// TIA Portal V17 export
// export: Created 2025-01-08T13:55:36.5022133Z, ExportSetting WithDefaults, DisplayName Totally Integrated Automation Portal, DisplayVersion V17, DisplayName TIA Portal Openness, DisplayVersion V17, DisplayName TIA Portal Version Control Interface, DisplayVersion V17, DisplayName SINAMICS Startdrive Advanced, DisplayVersion V17 Update2, DisplayName SINAMICS Startdrive G130, G150, S120, S150, SINAMICS MV, S210, DisplayVersion V17 Update2, DisplayName SINAMICS Startdrive G110M, G120, G120C, G120D, G120P, G115D, DisplayVersion V17 Update2, DisplayName STEP 7 Professional, DisplayVersion V17, DisplayName STEP 7 Safety, DisplayVersion V17, DisplayName WinCC Advanced, DisplayVersion V17
TYPE "HSMConfigAndMachineParameterMask"
// stored: IsFailsafeCompliant false
   STRUCT
      HSMConfig_1 : "HSMConfigParaMask1";
      HSMConfig_2 : "HSMConfigParaMask2";
      HSMMachine_1 { S7_SetPoint := 'True'} : "HSMMachineParaMask1";
      HSMMachine_2 { S7_SetPoint := 'True'} : "HSMMachineParaMask2";
      HSMMachine_3 { S7_SetPoint := 'True'} : "HSMMachineParaMask3";
      HSMMachine_4 { S7_SetPoint := 'True'} : "HSMMachineParaMask4";
      HSMMachine_5 { S7_SetPoint := 'True'} : "HSMMachineParaMask5";
      HSMMachine_6 { S7_SetPoint := 'True'} : "HSMMachineParaMask6";
      HSMMachine_7 { S7_SetPoint := 'True'} : "HSMMachineParaMask7";
      HSMMachine_8 { S7_SetPoint := 'True'} : "HSMMachineParaMask8";
   END_STRUCT;
END_TYPE
